(* CODESYS project motors_afag_coe.library
   Author: Miroslav Kozarev
   Placeholder: Motors_AFAG_CoE
   Title: Motors_AFAG_CoE
   Version: 0.1
   Description: Miroslav-Sashev@sensata.com
   Company: Sensata Technologies Bulgaria

Project tree, tasks and I/O mapping:
  libraries: Motors_DUTs, * (Sensata Technologies Bulgaria); Tc2_Standard, * (Beckhoff Automation GmbH); Tc3_LinMot, 1.1.0.0 (NTI AG)
  DUTs/
    Motors/
      AFAG/
        data type T_LM_Axis
        data type T_LM_DrvToPlc
  POUs/
    Motors/
      AFAG/
        Subs/
          LinMot/
            function block FB_LM_AxisControl [ST]
            function block FB_LM_MoveAbs [ST]
            function block FB_LM_MoveVelocity [ST]
            function block FB_LM_Stop [ST]
            function FN_LM_UptMCI_2 [ST]
        function block FB_ServoAxis_LinMot [ST]: A_GenOutput, A_Home, A_MoveAbsolute, A_MoveVelocity, A_ParseInput, A_ResetDone, A_SetMovementData
*)

// DUTs/Motors/AFAG/T_LM_Axis
TYPE T_LM_Axis : 
STRUCT
	PlcToDrv			AT %Q* :tstLM_PlcToDrv; 													(*PLC to Drive struct*)
	DrvToPlc			AT %I* :T_LM_DrvToPlc; 														(*Drive to PLC struct*)
	(*Status information*)
	AxisState			: tenLM_AxisState;
	CommandRunning		: BOOL;
	CommandAborted		: BOOL;
	ConfigChannelBusy	: BOOL;
	(*Information (Not required for prober work of the library function blocks)*)
	AxisName			: STRING;
	AxisNr				: UINT;
	AxisCtrlType		: STRING; 																	(*Eg. 'E1200-EC-UC', 'E1130-DP', 'B1100-GP', ....*)
END_STRUCT
END_TYPE

// DUTs/Motors/AFAG/T_LM_DrvToPlc
TYPE T_LM_DrvToPlc :
STRUCT
	StateVar 			: UINT; 																	(*StateVar of the drive*)
	StatusWord 			: UINT; 																	(*Statusword of the drive*)
	WarnWord 			: UINT; 																	(*Warnword of the drive*)
	ComDemandPosition 	: DINT; 																	(*32Bit demand position*)
	ComDemandVelocity	: DINT; 																	
	ComActualPosition 	: DINT; 																	(*32Bit actual position*)
	ComActualVelocity	: DINT; 																	

	CfgStatusWord 		: UINT;  																	(*Config Channel Status*)
	CfgIndexIn 			: UINT;  																	(*Argument (meaning depends on Cmd ID*)
	CfgValueIn 			: UDINT; 																	(*Argument (meaning depends on Cmd ID*)
END_STRUCT
END_TYPE

// POUs/Motors/AFAG/Subs/LinMot/FB_LM_AxisControl
FUNCTION_BLOCK FB_LM_AxisControl
VAR_INPUT
	SwitchOn		    : BOOL;	(*Switch on motor*)
	Home				: BOOL;	(*Start homing procedure*)
	ErrorAcknowledge	: BOOL;	(*Error acknowledge*)
	JogPlus				: BOOL;	(*Jog move postive*)
	JogMinus			: BOOL;	(*Jog move negative*)
	Band				: REAL := 10000;
END_VAR
VAR_IN_OUT
	Axis	       		: T_LM_Axis; (*Axis reference*)
END_VAR
VAR_OUTPUT
	OperationEnabled	: BOOL;	(*Axis powered on*)
	SwitchOnLocked		: BOOL;	(*Switch on locked*)
	Homed     	      	: BOOL;	(*Axis has reference*)
	MotionActive		: BOOL;	(*Motion active (Setpoint generation (VAI, curve) active)*)
	Jogging				: BOOL;	(*Axis is moving in jog mode*)
	Warning         	: BOOL;	(*Warning detected*)
	Error          		: BOOL;	(*Error detected*)
	ErrorCode      		: UINT;	(*Error code, see MotionCtrlSW manual*)
	DemandPosition  	: REAL;	(*Demand position in [mm]*)
	ActualPosition  	: REAL;	(*Actual position in [mm]*)
	ActualCurrent   	: REAL;	(*Actual motor current in [A]*)
	ActualVelocity		: REAL;
	DemandVelocity		: REAL;
END_VAR
VAR
	uiState        		: UINT;	(*internal -> Current state of the drive*)
	rTrigHome 			: LM_R_TRIG;	(*internal ->*)
	fTrigHome 			: LM_F_TRIG;	(*internal ->*)
END_VAR
(*Version history:
Date         	 | Version    		| Created under     	| Author          	| Remark 
------------------------------------------------------------------------------------------------------------------------------- 
2011-jul-12   	 | 1.0.0      		| V2.11.0 (Build 1016)	| fj  				| initial release 
2011-nov-22   	 | 1.0.1      		| V2.11.0 (Build 1016)	| fj  				| homed output reset if home input is set 
2011-dec-01   	 | 1.0.2      		| V2.11.0 (Build 1016)	| fj  				| code optimisation
2012-jan-25   	 | 1.0.3     		| V2.11.0 (Build 1016)	| fj  				| operation enabled output is now directly mapped to the status word bit 0
2012-oct-16   	 | 1.1.0      		| V2.11.0 (Build 1016)	| fj  				| added additional StateVar check for 090Fh ("homing finished") when rehoming
2014-may-13   	 | 1.0.0.1     		| v3.14014.0			| fj  				| added output DemandPosition
																				| optimized home input / homed output behaviour
*)

(*Eingänge zuweisen/lesen ][ Read and allocate inputs*)
	ActualPosition := DINT_TO_REAL(Axis.DrvToPlc.ComActualPosition)/Band;
	DemandPosition := DINT_TO_REAL(Axis.DrvToPlc.ComDemandPosition)/Band;
	ActualVelocity := DINT_TO_REAL(Axis.DrvToPlc.ComActualVelocity)/Band;
	DemandVelocity := DINT_TO_REAL(Axis.DrvToPlc.ComDemandVelocity)/Band;
	
	(*Workaround for different XML current definitions (16Bit/32Bit)*)
	//IF Axis.DrvToPlc.ComActualCurrent32 = 0 AND Axis.DrvToPlc.ComActualCurrent16 = 0 THEN
	//	ActualCurrent := 0;
	//ELSIF Axis.DrvToPlc.ComActualCurrent32 <> 0 AND Axis.DrvToPlc.ComActualCurrent16 = 0 THEN
	//	ActualCurrent := DINT_TO_REAL(Axis.DrvToPlc.ComActualCurrent32)/1000;
	//ELSIF Axis.DrvToPlc.ComActualCurrent32 = 0 AND Axis.DrvToPlc.ComActualCurrent16 <> 0 THEN
	//	ActualCurrent := INT_TO_REAL(Axis.DrvToPlc.ComActualCurrent16)/1000;
	//ELSE
	//	ActualCurrent := DINT_TO_REAL(Axis.DrvToPlc.ComActualCurrent32)/1000; (*If both 16/32Bit currents aren't 0 32Bit has higher priority*)
	//END_IF

(*Variablen ][ variables*)
	uiState := SHR(Axis.DrvToPlc.StateVar, 8);
	SwitchOnLocked := Axis.DrvToPlc.StatusWord.6;
	Warning := Axis.DrvToPlc.StatusWord.7;
	MotionActive := Axis.DrvToPlc.StatusWord.13;
	OperationEnabled := Axis.DrvToPlc.StatusWord.0;

(*=============================================================================
*  State Machine
===============================================================================*)    

CASE uiState OF
	(*Not Ready to Switch On*)
	00:	Axis.AxisState := Disabled_LM;

	(*State 4: Error*)
	04:	ErrorCode := UINT_TO_USINT(Axis.DrvToPlc.StateVar);
		Error := TRUE;
		Axis.AxisState := ErrorStop_LM;

	(*State 8: Operation Enabled*)
	08:	Homed := Axis.DrvToPlc.StateVar.7;
		IF Axis.DrvToPlc.StatusWord.13 AND NOT (Axis.AxisState = Stopping_LM) THEN
			Axis.AxisState := DiscreteMotion_LM;
		ELSIF NOT Axis.DrvToPlc.StatusWord.13 AND NOT (Axis.AxisState = Stopping_LM) THEN
			Axis.AxisState := StandStill_LM;
		END_IF

	(*State 9: Homing*)
	09:	Axis.AxisState := Homing_LM;
		IF Axis.DrvToPlc.StateVar = 16#090F THEN
			Axis.PlcToDrv.ControlWord.11 := FALSE;
		END_IF

	(*State 14: Error Behaviour QuickStop*)
	14:	Axis.AxisState := ErrorStop_LM;

	(*State 16: Jogging +*)
	16:	Axis.AxisState := Jogging_LM;

	(*State 17: Jogging -*)
	17:	Axis.AxisState := Jogging_LM;

END_CASE;


(*Wenn der drive nicht im Fehlerzustand ist, werden Error und ErrorCode auf Null gesetzt*)
(*If the drive is not in Error state, Error and ErrorCode are set to zero*)
IF uiState <> 16#04 THEN
	Error := FALSE;
	ErrorCode := 16#00;
END_IF;

IF uiState <> 16#08 THEN
	Axis.PlcToDrv.MCHeader := 16#0000; (*Reset Header to prevent "MC Cmd in wrong state" error*)
	Axis.CommandRunning := FALSE;
	Axis.CommandAborted := FALSE;
END_IF;

(*Switch On*)
Axis.PlcToDrv.ControlWord.0 := SwitchOn;
IF NOT Axis.PlcToDrv.ControlWord.0 AND NOT (uiState = 4 OR uiState = 14) THEN
	Axis.AxisState := Disabled_LM;
END_IF

(*Home*)
rTrigHome(CLK:=Home);
fTrigHome(CLK:=Home);
IF rTrigHome.Q THEN
	Axis.PlcToDrv.ControlWord.11 := TRUE;
END_IF
IF fTrigHome.Q  THEN
	Axis.PlcToDrv.ControlWord.11 := FALSE;
END_IF

IF uiState = 16#09 OR (Axis.PlcToDrv.ControlWord.11 AND NOT (uistate = 16#09)) THEN
	Homed := FALSE;
ELSE
	Homed := Axis.DrvToPlc.StatusWord.11;
END_IF

(*Error acknowledge*)
Axis.PlcToDrv.ControlWord.7 := ErrorAcknowledge;

(*JogPlus*)
Axis.PlcToDrv.ControlWord.8 := JogPlus;

(*JogMinus*)
Axis.PlcToDrv.ControlWord.9 := JogMinus;

IF (uiState = 16 OR uiState = 17) AND UINT_TO_USINT(Axis.DrvToPlc.StateVar) = 16#01 THEN
	Jogging := TRUE;
ELSE
	Jogging := FALSE;
END_IF

END_FUNCTION_BLOCK

// POUs/Motors/AFAG/Subs/LinMot/FB_LM_MoveAbs
FUNCTION_BLOCK FB_LM_MoveAbs
VAR_INPUT
	Execute			:BOOL;	(*Execute command*)
	Position		:REAL;	(*Target position in [mm]*)
	Velocity		:REAL;	(*Maximal velocity in [m/s]*)
	Acceleration	:REAL;	(*Acceleration in [m/s^2]*)
	Deceleration	:REAL;	(*Deceleration in [m/s^2]*)
	Band			: REAL := 10000;
END_VAR
VAR_IN_OUT
	Axis			:T_LM_Axis; (*Axis reference*)
	bResetDone		:BOOL;
END_VAR
VAR_OUTPUT
	Done			:BOOL;	(*Command has been executed*)
	Busy			:BOOL;	(*Command running / FB Busy*)
	Error			:BOOL;	(*Error detected*)
	ErrorID			:UINT;	(*Error ID:
							01h: Axis not ready
 							02h: Axis already has command running
 							03h: Axis has error
 							04h: Command interrupted
 							05h: Command aborted
							06h: Invalid input(s)
							*)
END_VAR

VAR_IN_OUT
	
END_VAR

VAR
	usiOldCmdCount 	:USINT;	(*internal -> *)
	usiNewCmdCount	:USINT;	(*internal -> *)
	uiCState		:UINT;	(*internal -> *)
	uiFbState		:UINT;	(*internal -> *)
	rTrig			:LM_R_TRIG;	(*internal -> *)
	udiTmpDWord		:UDINT;	(*internal -> *)

 	uiCmdHeader 	:UINT := 16#0100;	(*CommandHeader (010xh) of the "VAI Go To Position (010xh)" motion command*)
END_VAR
(*Version history:
Date         	 | Version    		| Created under     	| Author          	| Remark 
------------------------------------------------------------------------------------------------------------------------------- 
2011-jul-12   	 | 1.0.0      		| V2.11.0 (Build 1016)	| fj  				| initial release 
2011-sep-13   	 | 1.0.1      		| V2.11.0 (Build 1016)	| fj  				| removed check on "StandStill_LM"
2011-dec-01   	 | 1.0.2      		| V2.11.0 (Build 1016)	| fj  				| code optimisation
2012-apr-25   	 | 1.1.0     		| V2.11.0 (Build 1016)	| fj  				| added input parameters check
*)

(*Variablen ][ variables*)
usiOldCmdCount := SHR(UINT_TO_USINT(SHL(Axis.DrvToPlc.StateVar,4)),4);
uiCState := SHR(Axis.DrvToPlc.StateVar, 8);

IF bResetDone THEN
	Done := FALSE;
	bResetDone := FALSE;
END_IF

(*Flankenerkennung am Execute Eingang*)
(*Edge detection on Execute input*)
rTrig(CLK:=Execute);
IF rTrig.Q AND uiCState = 16#08 AND NOT Axis.CommandRunning THEN (*Start command*)
	Axis.CommandRunning := TRUE;
	Busy := TRUE;
	Done := FALSE;
	uiFbState := 1;
ELSIF rTrig.Q AND Busy THEN (*Restart command / New rising edge on execute input*)
	Axis.CommandRunning := TRUE;
	Done := FALSE;
	Busy := TRUE;
	uiFbState := 1;
ELSIF rTrig.Q AND uiCState <> 16#08 THEN (*Axis not ready*)
	uiFbState := 50; (*Error state*)
	Done := FALSE;
	Error := TRUE;
	ErrorID := 16#01; (*Axis not ready*)
ELSIF rTrig.Q AND Axis.CommandRunning AND NOT Busy THEN (*Axis already has a command running*)
	uiFbState := 50; (*Error state*)
	Error := TRUE;
	ErrorID := 16#02; (*Axis already has a command running*)
END_IF

IF Busy AND uiCState = 16#04 THEN
	Axis.CommandRunning := FALSE;
	uiFbState := 50;
	Error := TRUE;
	ErrorID := 16#03; (*Axis has error*)
END_IF

IF Busy AND uiCState <> 16#08 THEN
	Axis.CommandRunning := FALSE;
	uiFbState := 50; (*Error state*)
	Error := TRUE;
	ErrorID := 16#04; (*Command interupted*)
ELSIF Busy AND Axis.CommandAborted THEN
	uiFbState := 50; (*Error state*)
	Error := TRUE;
	ErrorID := 16#05; (*Command aborted*)
END_IF

(*State machine*)
CASE uiFbState OF
	0:	;

	1:	(*Check inputs on valid value*)
		IF (-214748.0 <= Position AND Position <= 214748.0)
			AND (0.0 < Velocity AND Velocity <= 2147.0)
			AND (0.0 < Acceleration AND Acceleration <= 21474.0)
			AND (0.0 < Deceleration AND Deceleration <= 21474.0)
			THEN
			(*Befehlskopf mit CMD Count berechen und senden ][ Calculate and send command header*)
			usiNewCmdCount := (usiOldCmdCount + 1) MOD 16 ; (*MOD 16*)
			Axis.PlcToDrv.MCHeader := 16#0000; (*Reset Header*)
			Axis.PlcToDrv.MCHeader := uiCmdHeader + usiNewCmdCount;

			udiTmpDWord := DINT_TO_UDINT(REAL_TO_DINT(Position * Band)); (*Target position*)
			Axis.PlcToDrv.MCParaWord0 := UDINT_TO_UINT(udiTmpDWord);
			Axis.PlcToDrv.MCParaWord1 := UDINT_TO_UINT(ROR(udiTmpDWord,16));

			udiTmpDWord := DINT_TO_UDINT(REAL_TO_DINT(Velocity * 100 * Band)); (*Maximal velocity*)
			Axis.PlcToDrv.MCParaWord2 := UDINT_TO_UINT(udiTmpDWord);
			Axis.PlcToDrv.MCParaWord3 := UDINT_TO_UINT(ROR(udiTmpDWord,16));

			udiTmpDWord := DINT_TO_UDINT(REAL_TO_DINT(Acceleration * 10 * Band)); (*Acceleration*)
			Axis.PlcToDrv.MCParaWord4 := UDINT_TO_UINT(udiTmpDWord);
			Axis.PlcToDrv.MCParaWord5 := UDINT_TO_UINT(ROR(udiTmpDWord,16));

			udiTmpDWord := DINT_TO_UDINT(REAL_TO_DINT(Deceleration * 10 * Band)); (*Deceleration*)
			Axis.PlcToDrv.MCParaWord6 := UDINT_TO_UINT(udiTmpDWord);
			Axis.PlcToDrv.MCParaWord7 := UDINT_TO_UINT(ROR(udiTmpDWord,16));

			FN_LM_UptMCI_2(Axis);
			
			uiFbState := 2;
		ELSE
			Axis.CommandRunning := FALSE;
			uiFbState := 50; (*Error state*)
			Error := TRUE;
			ErrorID := 16#06; (*Invalid input(s)*)
		END_IF

	2:	(*Prüfen ob Befehl ausgeführt ][ Check if command has been executed*)
		IF usiOldCmdCount = usiNewCmdCount AND uiCState = 16#08 AND Axis.DrvToPlc.StateVar.6 THEN
			Done := TRUE;
			Busy := FALSE;
			Axis.PlcToDrv.MCHeader := 16#0000 + usiNewCmdCount; (*Send no operation*)
			Axis.CommandRunning := FALSE;
			uiFbState := 3;
		END_IF

	3:	IF NOT Execute THEN
			uiFbState := 0;
			Busy := FALSE;
		END_IF

	50:	Error := TRUE;
		Busy := FALSE;
		Done := FALSE;
		IF NOT Execute THEN
			uiFbState := 0;
			Error := FALSE;
			ErrorID := 0;
		END_IF

END_CASE

END_FUNCTION_BLOCK

// POUs/Motors/AFAG/Subs/LinMot/FN_LM_UptMCI_2
FUNCTION FN_LM_UptMCI_2 : BOOL
VAR_IN_OUT
	Axis 	:T_LM_Axis;
END_VAR
VAR
END_VAR

Axis.PlcToDrv.MCParaDWord_00_03 := SHL(UINT_TO_UDINT(Axis.PlcToDrv.MCParaWord1),16) + UINT_TO_UDINT(Axis.PlcToDrv.MCParaWord0);
Axis.PlcToDrv.MCParaDWord_04_07 := SHL(UINT_TO_UDINT(Axis.PlcToDrv.MCParaWord3),16) + UINT_TO_UDINT(Axis.PlcToDrv.MCParaWord2);
Axis.PlcToDrv.MCParaDWord_08_11 := SHL(UINT_TO_UDINT(Axis.PlcToDrv.MCParaWord5),16) + UINT_TO_UDINT(Axis.PlcToDrv.MCParaWord4);
Axis.PlcToDrv.MCParaDWord_12_15 := SHL(UINT_TO_UDINT(Axis.PlcToDrv.MCParaWord7),16) + UINT_TO_UDINT(Axis.PlcToDrv.MCParaWord6);
Axis.PlcToDrv.MCParaDWord_16_19 := SHL(UINT_TO_UDINT(Axis.PlcToDrv.MCParaWord9),16) + UINT_TO_UDINT(Axis.PlcToDrv.MCParaWord8);
Axis.PlcToDrv.MCParaDWord_20_23 := SHL(UINT_TO_UDINT(Axis.PlcToDrv.MCParaWord11),16) + UINT_TO_UDINT(Axis.PlcToDrv.MCParaWord10);
Axis.PlcToDrv.MCParaDWord_24_27 := SHL(UINT_TO_UDINT(Axis.PlcToDrv.MCParaWord13),16) + UINT_TO_UDINT(Axis.PlcToDrv.MCParaWord12);

END_FUNCTION

// POUs/Motors/AFAG/Subs/LinMot/FB_LM_MoveVelocity
FUNCTION_BLOCK FB_LM_MoveVelocity
VAR_INPUT
	Execute					: BOOL;																	(*Execute command*)
	Velocity				: REAL;																	(*Maximal velocity in [m/s]*)
	Acceleration			: REAL;																	(*Acceleration in [m/s^2]*)
	NegativeDirection		: BOOL := FALSE;
	Band					: REAL := 10000;
	TargetReached			: BOOL;
END_VAR
VAR_IN_OUT
	Axis					: T_LM_Axis; 															(*Axis reference*)
END_VAR
VAR_OUTPUT
	Done					: BOOL;																	(*Command has been executed*)
	Busy					: BOOL;																	(*Command running / FB Busy*)
	Error					: BOOL;																	(*Error detected*)
	ErrorID					: UINT;																	(*Error ID:
																									01h: Axis not ready
 																									02h: Axis already has command running
 																									03h: Axis has error
 																									04h: Command interrupted
 																									05h: Command aborted
																									06h: Invalid input(s)
																									*)
END_VAR
VAR
	usiOldCmdCount 			: USINT;																(*internal -> *)
	usiNewCmdCount			: USINT;																(*internal -> *)
	uiCState				: UINT;																	(*internal -> *)
	uiFbState				: UINT;																	(*internal -> *)
	rTrig					: LM_R_TRIG;															(*internal -> *)
	udiTmpDWord				: UDINT;																(*internal -> *)

 	uiCmdHeader 			: UINT := 16#0CE0;														(*CommandHeader (0CExh) of the "VAI Dec=AccVAI Infinite Motion Positive Direction (0CExh)" motion command*)
END_VAR
(*Version history:
Date         	 | Version    		| Created under     	| Author          	| Remark 
------------------------------------------------------------------------------------------------------------------------------- 
2011-jul-12   	 | 1.0.0      		| V2.11.0 (Build 1016)	| fj  				| initial release 
2011-sep-13   	 | 1.0.1      		| V2.11.0 (Build 1016)	| fj  				| removed check for "StandStill_LM" on Execute rising edge
2011-dec-01   	 | 1.0.2      		| V2.11.0 (Build 1016)	| fj  				| code optimisation
2012-apr-25   	 | 1.1.0     		| V2.11.0 (Build 1016)	| fj  				| added input parameters check
*)

(*Variablen ][ variables*)
usiOldCmdCount := SHR(UINT_TO_USINT(SHL(Axis.DrvToPlc.StateVar,4)),4);
uiCState := SHR(Axis.DrvToPlc.StateVar, 8);

(*Flankenerkennung am Execute Eingang*)
(*Edge detection on Execute input*)
rTrig(CLK:=Execute);
IF rTrig.Q AND uiCState = 16#08 AND NOT Axis.CommandRunning THEN (*Start command*)
	Axis.CommandRunning := TRUE;
	Busy := TRUE;
	uiFbState := 1;
ELSIF rTrig.Q AND Busy THEN (*Restart command / New rising edge on execute input*)
	Axis.CommandRunning := TRUE;
	Busy := TRUE;
	uiFbState := 1;
ELSIF rTrig.Q AND uiCState <> 16#08 THEN (*Axis not ready*)
	uiFbState := 50; (*Error state*)
	Error := TRUE;
	ErrorID := 16#01; (*Axis not ready*)
ELSIF rTrig.Q AND Axis.CommandRunning AND NOT Busy THEN (*Axis already has a command running*)
	uiFbState := 50; (*Error state*)
	Error := TRUE;
	ErrorID := 16#02; (*Axis already has a command running*)
END_IF

IF Busy AND uiCState = 16#04 THEN
	Axis.CommandRunning := FALSE;
	uiFbState := 50;
	Error := TRUE;
	ErrorID := 16#03; (*Axis has error*)
END_IF

IF Busy AND uiCState <> 16#08 THEN
	Axis.CommandRunning := FALSE;
	uiFbState := 50; (*Error state*)
	Error := TRUE;
	ErrorID := 16#04; (*Command interupted*)
ELSIF Busy AND Axis.CommandAborted THEN
	uiFbState := 50; (*Error state*)
	Error := TRUE;
	ErrorID := 16#05; (*Command aborted*)
END_IF

(*State machine*)
CASE uiFbState OF
	0:	;

	1:	(*Check inputs on valid value*)
		IF (-10.0 <= ABS(Velocity) AND ABS(Velocity) <= 99999999)
			AND (0.0 < Acceleration AND Acceleration <= 99999999)
			THEN
			(*Befehlskopf mit CMD Count berechen und senden ][ Calculate and send command header*)
			usiNewCmdCount := (usiOldCmdCount + 1) MOD 16 ; (*MOD 16*)
			Axis.PlcToDrv.MCHeader := 16#0000; (*Reset Header*)
			NegativeDirection := Velocity < 0;
			IF NegativeDirection THEN
 				uiCmdHeader := 16#0CF0;
			ELSE
 				uiCmdHeader := 16#0CE0;
			END_IF
			
			Axis.PlcToDrv.MCHeader := uiCmdHeader + usiNewCmdCount;

			udiTmpDWord := DINT_TO_UDINT(REAL_TO_DINT(ABS(Velocity) * 100 * Band)); (*Maximal velocity*)
			Axis.PlcToDrv.MCParaWord0 := UDINT_TO_UINT(udiTmpDWord);
			Axis.PlcToDrv.MCParaWord1 := UDINT_TO_UINT(ROR(udiTmpDWord,16));

			udiTmpDWord := DINT_TO_UDINT(REAL_TO_DINT(Acceleration * 10000)); (*Acceleration / Deceleration*)
			Axis.PlcToDrv.MCParaWord2 := UDINT_TO_UINT(udiTmpDWord);
			Axis.PlcToDrv.MCParaWord3 := UDINT_TO_UINT(ROR(udiTmpDWord,16));
			FN_LM_UptMCI_2(Axis);

			uiFbState := 2;
		ELSE
			Axis.CommandRunning := FALSE;
			uiFbState := 50; (*Error state*)
			Error := TRUE;
			ErrorID := 16#06; (*Invalid input(s)*)
		END_IF

	2:	(*Prüfen ob Befehl ausgeführt ][ Check if command has been executed*)
		IF (usiOldCmdCount = usiNewCmdCount AND uiCState = 16#08 AND TargetReached) (*Axis.DrvToPlc.StateVar.6) OR
			TargetReached*) THEN
			Done := TRUE;
			Busy := FALSE;
			Axis.PlcToDrv.MCHeader := 16#0000 + usiNewCmdCount; (*Send no operation*)
			Axis.CommandRunning := FALSE;
			uiFbState := 3;
		END_IF

	3:	IF NOT Execute THEN
			uiFbState := 0;
			Busy := FALSE;
			Done := FALSE;
		END_IF

	50:	Error := TRUE;
		Busy := FALSE;
		Done := FALSE;
		IF NOT Execute THEN
			uiFbState := 0;
			Error := FALSE;
			ErrorID := 0;
		END_IF

END_CASE

END_FUNCTION_BLOCK

// POUs/Motors/AFAG/Subs/LinMot/FB_LM_Stop
FUNCTION_BLOCK FB_LM_Stop
VAR_INPUT
	Execute					: BOOL;																	(*Execute command*)
	Velocity				: REAL;																	(*Maximal velocity in [m/s]*)
	Acceleration			: REAL;																	(*Acceleration in [m/s^2]*)
	NegativeDirection		: BOOL := FALSE;
	Band					: REAL := 10000;
	TargetReached			: BOOL;
END_VAR
VAR_IN_OUT
	Axis					: T_LM_Axis; 															(*Axis reference*)
END_VAR
VAR_OUTPUT
	Done					: BOOL;																	(*Command has been executed*)
	Busy					: BOOL;																	(*Command running / FB Busy*)
	Error					: BOOL;																	(*Error detected*)
	ErrorID					: UINT;																	(*Error ID:
																									01h: Axis not ready
 																									02h: Axis already has command running
 																									03h: Axis has error
 																									04h: Command interrupted
 																									05h: Command aborted
																									06h: Invalid input(s)
																									*)
END_VAR
VAR
	usiOldCmdCount 			: USINT;																(*internal -> *)
	usiNewCmdCount			: USINT;																(*internal -> *)
	uiCState				: UINT;																	(*internal -> *)
	uiFbState				: UINT;																	(*internal -> *)
	rTrig					: LM_R_TRIG;															(*internal -> *)
	udiTmpDWord				: UDINT;																(*internal -> *)

 	uiCmdHeader 			: UINT := 16#0170;														(*CommandHeader (0CExh) of the "VAI Dec=AccVAI Infinite Motion Positive Direction (0CExh)" motion command*)
END_VAR
(*Version history:
Date         	 | Version    		| Created under     	| Author          	| Remark 
------------------------------------------------------------------------------------------------------------------------------- 
2011-jul-12   	 | 1.0.0      		| V2.11.0 (Build 1016)	| fj  				| initial release 
2011-sep-13   	 | 1.0.1      		| V2.11.0 (Build 1016)	| fj  				| removed check for "StandStill_LM" on Execute rising edge
2011-dec-01   	 | 1.0.2      		| V2.11.0 (Build 1016)	| fj  				| code optimisation
2012-apr-25   	 | 1.1.0     		| V2.11.0 (Build 1016)	| fj  				| added input parameters check
*)

(*Variablen ][ variables*)
usiOldCmdCount := SHR(UINT_TO_USINT(SHL(Axis.DrvToPlc.StateVar,4)),4);
uiCState := SHR(Axis.DrvToPlc.StateVar, 8);

(*Flankenerkennung am Execute Eingang*)
(*Edge detection on Execute input*)
rTrig(CLK:=Execute);
IF rTrig.Q AND uiCState = 16#08 AND NOT Axis.CommandRunning THEN (*Start command*)
	Axis.CommandRunning := TRUE;
	Busy := TRUE;
	uiFbState := 1;
ELSIF rTrig.Q AND Busy THEN (*Restart command / New rising edge on execute input*)
	Axis.CommandRunning := TRUE;
	Busy := TRUE;
	uiFbState := 1;
ELSIF rTrig.Q AND uiCState <> 16#08 THEN (*Axis not ready*)
	uiFbState := 50; (*Error state*)
	Error := TRUE;
	ErrorID := 16#01; (*Axis not ready*)
ELSIF rTrig.Q AND Axis.CommandRunning AND NOT Busy THEN (*Axis already has a command running*)
	uiFbState := 50; (*Error state*)
	Error := TRUE;
	ErrorID := 16#02; (*Axis already has a command running*)
END_IF

IF Busy AND uiCState = 16#04 THEN
	Axis.CommandRunning := FALSE;
	uiFbState := 50;
	Error := TRUE;
	ErrorID := 16#03; (*Axis has error*)
END_IF

IF Busy AND uiCState <> 16#08 THEN
	Axis.CommandRunning := FALSE;
	uiFbState := 50; (*Error state*)
	Error := TRUE;
	ErrorID := 16#04; (*Command interupted*)
ELSIF Busy AND Axis.CommandAborted THEN
	uiFbState := 50; (*Error state*)
	Error := TRUE;
	ErrorID := 16#05; (*Command aborted*)
END_IF

(*State machine*)
CASE uiFbState OF
	0:	;

	1:	(*Check inputs on valid value*)
		IF (0.0 < Acceleration AND Acceleration <= 99999999)
			THEN
			(*Befehlskopf mit CMD Count berechen und senden ][ Calculate and send command header*)
			usiNewCmdCount := (usiOldCmdCount + 1) MOD 16 ; (*MOD 16*)
			Axis.PlcToDrv.MCHeader := 16#0000; (*Reset Header*)
			
			uiCmdHeader := 16#0170;
			
			Axis.PlcToDrv.MCHeader := uiCmdHeader + usiNewCmdCount;

			udiTmpDWord := DINT_TO_UDINT(REAL_TO_DINT(Acceleration * 10000)); (*Acceleration / Deceleration*)
			Axis.PlcToDrv.MCParaWord0 := UDINT_TO_UINT(udiTmpDWord);
			Axis.PlcToDrv.MCParaWord1 := UDINT_TO_UINT(ROR(udiTmpDWord,16));
			FN_LM_UptMCI_2(Axis);

			uiFbState := 2;
		ELSE
			Axis.CommandRunning := FALSE;
			uiFbState := 50; (*Error state*)
			Error := TRUE;
			ErrorID := 16#06; (*Invalid input(s)*)
		END_IF

	2:	(*Prüfen ob Befehl ausgeführt ][ Check if command has been executed*)
		IF (usiOldCmdCount = usiNewCmdCount AND uiCState = 16#08 AND TargetReached) (*Axis.DrvToPlc.StateVar.6) OR
			TargetReached*) THEN
			Done := TRUE;
			Busy := FALSE;
			Axis.PlcToDrv.MCHeader := 16#0000 + usiNewCmdCount; (*Send no operation*)
			Axis.CommandRunning := FALSE;
			uiFbState := 3;
		END_IF

	3:	IF NOT Execute THEN
			uiFbState := 0;
			Busy := FALSE;
			Done := FALSE;
		END_IF

	50:	Error := TRUE;
		Busy := FALSE;
		Done := FALSE;
		IF NOT Execute THEN
			uiFbState := 0;
			Error := FALSE;
			ErrorID := 0;
		END_IF

END_CASE

END_FUNCTION_BLOCK

// POUs/Motors/AFAG/FB_ServoAxis_LinMot
FUNCTION_BLOCK FB_ServoAxis_LinMot																	// HJ LinMot Afaq - use with older controllers in combination with Tc3_LinMot library.
VAR_INPUT
	IsAbsolute						: BOOL := FALSE;												// Use to mark that the axis is with an absolute encoder and no homing should be executed.
	InvertMotorPolarity				: BOOL := FALSE;												// Use this to invert the motor encoder polarity from here. (CurrentPosition or TargetPosition * -1 FTW)
	Band							: REAL := 10000;												// Encoder multiplier.
	DoStop							: BOOL;															// NOT WORKING!!!
END_VAR
VAR_OUTPUT
	CurrentPosition					: LREAL;														// The current motor position.
	CurrentCommand					: UDINT;														// The current motor command.
	CurrentVelocity			 		: LREAL;														// The current motor velocity.
	Enabled							: BOOL;															// Is the motor enabled for operation.
	Error							: BOOL;															// Is the motor in an error state.
	ErrorID							: UDINT;														// If the motor is in an error state this will hold the error data.
	Moving							: BOOL;															// Is the motor moving.	
	Refferenced 					: BOOL;															// Is the motor referenced - homed.
	TraveledPath					: LREAL;														// The motor last traveled path. Currently valid only when in positioning mode.
	Busy							: BOOL;															// Is the motor busy - executing command.
	Stopped							: BOOL;															// Is the motor stopped - not working.
END_VAR
VAR_IN_OUT
	// As a test
	TargetPosition					: REAL;															// The target position of the motor. If DoMove is set in the right conditions, this will be sent to the motor.
	TargetVelocity					: REAL;															// The motor target movement velocity.
	TargetAcceleration				: REAL;															// The motor target acceleration.
	TargetDeceleration				: REAL;															// The motor target deceleration.
	TargetPrecision					: REAL;															// The motor target precision. Could use this dynamically troughout different states when the precision needs change.
	OperationMode					: UDINT := 0;													// The motor target operation mode 0 - Positioning, 1 - Velocity.
	DoServoOn						: BOOL;															// Activate the motor power up.
	DoReset							: BOOL;															// Activate the motor reset.
	DoHome							: BOOL;															// Activate the motor homing function. If the motor is marked as an absolute one this will only be reset and no homing will take place.
	DoMove							: BOOL;															// Activate a movement command. The values set in the TargetPosition, TargetVelocity and TargetAcceleration will be sent to the motor.
	TargetReached					: BOOL;															// Is the motor target reached in both modes (The target position or velocity is reached).
	axis							: T_LM_Axis;													// Lin Mot Axis reference - the actual IO structure. - LINMOT Legacy type T_LM_Axis.
END_VAR
VAR		
	state							: E_MotorStates;												// Current motor function block state.
	fbTimer							: TON;															// Used for timeouts and etc..
	fbResetTimer					: TON;															// Used for reset timeout.
	fbMoveAbsolute					: FB_LM_MoveAbs;												// Move absolute function block										- LINMOT Legacy type FB_LM_MoveAbs.
	fbMoveVelocity					: FB_LM_MoveVelocity;											// Move to velocity function block.
	fbAxisControl					: FB_LM_AxisControl;											// Axis control function block 										- LINMOT Legacy type FB_LM_AxisControl.
	fbAxisStop						: FB_LM_Stop;													// Axis stop function block.
	fbTriggerF						: F_TRIG;														// Disable trigger.
	
	PositioningMovement				: BOOL;
	VelocityMovement				: BOOL;
	
	bResetDone						: BOOL 							:= FALSE;						// Use to reset the done flag within the fbMoveAbsolute block.
	TargetTravelPath				: LREAL;														// Used to hold the target travel path.
	VelocityReached					: BOOL;
	VelocityMonitorDelimiter		: LREAL := 1000;
	TargetedVelocity				: LREAL;
	MovingToPositiong				: BOOL;
	MovingWithVelocity				: BOOL;
	MotionActive					: BOOL;
	EngageAxisStop					: BOOL;
	AxisStopping					: BOOL;
	AxisStopped						: BOOL;
	
	StopState						: DINT := 0;
	
	NegativeDirection				: BOOL := FALSE;
END_VAR

/////////////////////////////////////////////////
// NB!!!
// SET Acceleration/Deceleration at least once due to value checker. 
// 
// - prepared within the start movement state with A_SetMovementData();
//
/////////////////////////////////////////////////

//===============================================================

IF InvertMotorPolarity THEN
	TargetPosition := TargetPosition * -1;
END_IF

A_ParseInput();

fbTriggerF(CLK := DoServoOn);
		
IF fbTriggerF.Q AND 
	(state <> E_MotorStates.MOTORSTATE_ERROR) THEN
	state := E_MotorStates.MOTORSTATE_INIT;		
END_IF

IF (state <> E_MotorStates.MOTORSTATE_ERROR) AND 
	(state <> E_MotorStates.MOTORSTATE_RESET) AND 
	(state <> E_MotorStates.MOTORSTATE_ENABLE) AND 
	(DoReset = TRUE) THEN
	state := E_MotorStates.MOTORSTATE_RESET;
	IF DoMove OR 
		fbMoveAbsolute.Execute OR
		PositioningMovement OR 
		fbMoveVelocity.Execute OR
		VelocityMovement THEN
		DoMove := FALSE;
		PositioningMovement := FALSE;
		fbMoveAbsolute.Execute := FALSE;
		VelocityMovement := FALSE;
		fbMoveVelocity.Execute := FALSE;
	END_IF
	DoReset := FALSE;
END_IF

CASE state OF
	E_MotorStates.MOTORSTATE_INIT:
		DoMove := FALSE;
		PositioningMovement := FALSE;
		VelocityMovement := FALSE;
		DoHome := FALSE;
		A_ResetDone();
		DoServoOn := FALSE;
		DoReset := FALSE;
		state := E_MotorStates.MOTORSTATE_ENABLE;
		
	E_MotorStates.MOTORSTATE_ENABLE:
		IF Enabled THEN
			state := E_MotorStates.MOTORSTATE_OPERATIONAL;
		ELSIF Error OR DoReset THEN
			state := E_MotorStates.MOTORSTATE_RESET;
		END_IF
		
	E_MotorStates.MOTORSTATE_OPERATIONAL:
		IF fbTriggerF.Q THEN
			state := E_MotorStates.MOTORSTATE_INIT;	
		ELSE
			IF Error THEN
				DoServoOn := FALSE;
				state := E_MotorStates.MOTORSTATE_ERROR;
			ELSE
				IF DoMove THEN
					CASE OperationMode OF
						
						0:
							TargetReached := FALSE;
							TargetTravelPath := TargetPosition - CurrentPosition;
							A_ResetDone();
							A_SetMovementData();
							TargetedVelocity := TargetVelocity;
							//PositioningMovement := TRUE;
							StopState := 0;
							state := E_MotorStates.MOTORSTATE_MOVING;	
							
						1:
							TargetReached := FALSE;
							A_ResetDone();
							//VelocityMovement := TRUE;
							TargetedVelocity := TargetVelocity;
							NegativeDirection := TargetedVelocity < 0;
							StopState := 0;
							state := E_MotorStates.MOTORSTATE_MOVING_VELOCITY;
							
						ELSE
							
							state := E_MotorStates.MOTORSTATE_ERROR;
							
					END_CASE
				ELSIF DoHome THEN
					IF IsAbsolute THEN
						DoHome := FALSE;
					ELSE
						A_ResetDone();
						state := E_MotorStates.MOTORSTATE_HOMING;
					END_IF
				END_IF
			END_IF
		END_IF
		
	E_MotorStates.MOTORSTATE_MOVING:
		A_MoveAbsolute();
		
	E_MotorStates.MOTORSTATE_MOVING_VELOCITY:
		A_MoveVelocity();
		
	E_MotorStates.MOTORSTATE_HOMING:
		A_Home();
		
	E_MotorStates.MOTORSTATE_STOP:
		IF DoStop THEN
			EngageAxisStop := TRUE;
			fbAxisStop.Acceleration := TargetAcceleration;
			IF AxisStopped THEN
				Stopped := TRUE;
			END_IF
		ELSE
			EngageAxisStop := FALSE;
			Stopped := FALSE;
			state := E_MotorStates.MOTORSTATE_ENABLE;
		END_IF
		
	E_MotorStates.MOTORSTATE_ERROR:
		IF DoReset THEN
			IF Error THEN
				state := E_MotorStates.MOTORSTATE_RESET;
			ELSE
				state := E_MotorStates.MOTORSTATE_INIT;
			END_IF	
		END_IF
		
	E_MotorStates.MOTORSTATE_RESET:
		fbResetTimer(IN := TRUE, 
			PT := T#300MS);
		IF (NOT Error) THEN
			fbResetTimer(IN := FALSE);
			state := E_MotorStates.MOTORSTATE_INIT;
		ELSIF fbResetTimer.Q THEN
			fbResetTimer(IN := FALSE);
			DoReset := FALSE;
			state := E_MotorStates.MOTORSTATE_ERROR;
		END_IF

END_CASE

fbAxisControl(SwitchOn 					:= DoServoOn,
				Home 					:= DoHome, 
				ErrorAcknowledge 		:= DoReset,
				OperationEnabled 		=> Enabled,
				Homed 					=> Refferenced,
				MotionActive 			=> MotionActive,
				Error 					=> Error,
				ErrorCode 				=> ErrorID,
				ActualPosition 			=> CurrentPosition,
				//ActualVelocity 			=> CurrentVelocity,
				Axis 					:= axis);
				
fbMoveAbsolute(Axis 					:= axis,
				Execute 				:= PositioningMovement,
				Band					:= Band,
				Busy 					=> MovingToPositiong,
				Done 					=> TargetReached,
				bResetDone 				:= bResetDone);
				
fbAxisStop(Axis							:= axis,
	
				Execute					:= EngageAxisStop,
				
				Busy					=> AxisStopping,
				Done					=> AxisStopped);
				
				
IF OperationMode = 1 THEN
	A_GenOutput();
END_IF

fbMoveVelocity(Axis						:= axis,
				Execute					:= VelocityMovement,
				Band					:= Band,
				TargetReached			:= OperationMode = 1 AND TargetReached,
				Busy					=> MovingWithVelocity,
				Done					=> VelocityReached);
				
A_GenOutput();

IF OperationMode = 0 THEN
	Moving := MovingToPositiong OR MotionActive;
ELSE
	Moving := (ABS(CurrentVelocity) > 10) OR MovingWithVelocity;
END_IF

IF InvertMotorPolarity THEN
	CurrentPosition := CurrentPosition * -1;
END_IF

ACTION A_GenOutput:

IF VelocityMonitorDelimiter > 0 THEN
	CurrentVelocity := axis.DrvToPlc.ComActualVelocity / VelocityMonitorDelimiter;
END_IF

IF TargetPrecision > 0.0001 THEN
	IF OperationMode = 0 THEN
		TargetReached := TargetReached AND 
			(ABS(CurrentPosition - TargetPosition) < TargetPrecision) AND
			(NOT DoMove) AND
			(NOT PositioningMovement) AND
			(NOT DoStop);
	ELSIF OperationMode = 1 THEN
		IF ABS(TargetedVelocity) > 10 THEN
			TargetReached := ABS(TargetedVelocity - CurrentVelocity) < (ABS(TargetedVelocity) * (TargetPrecision / 100));
		ELSE
			TargetReached := ABS(TargetedVelocity - CurrentVelocity) < 10;
		END_IF
	END_IF
ELSE
	TargetReached := TargetReached AND 
		(ABS(CurrentPosition - TargetPosition) < 0.03) AND
		(NOT DoMove) AND
		(NOT PositioningMovement);
END_IF
END_ACTION

ACTION A_Home:
// Engage homing sequence.
IF Refferenced THEN
	DoHome := FALSE;
	state := E_MotorStates.MOTORSTATE_ENABLE;
ELSE
	IF Error THEN
		DoHome := FALSE;
		state := E_MotorStates.MOTORSTATE_ERROR;		
	END_IF
END_IF
END_ACTION

ACTION A_MoveAbsolute:
// Engage movement sequence.
IF NOT DoStop THEN
	A_SetMovementData();
END_IF
PositioningMovement := TRUE;
fbMoveAbsolute.Execute := PositioningMovement;
Busy := TRUE;
IF fbMoveAbsolute.Done AND
	(NOT DoStop) THEN
	Busy := FALSE;
	DoMove := FALSE;
	PositioningMovement := FALSE;
	fbMoveAbsolute.Execute := DoMove; 
	TraveledPath := TargetTravelPath;
	state := E_MotorStates.MOTORSTATE_ENABLE;
ELSIF fbMoveAbsolute.Error THEN
	DoMove := FALSE;
	PositioningMovement := FALSE;
	fbMoveAbsolute.Execute := DoMove;
	IF fbMoveAbsolute.ErrorID = 16#06 THEN			// BAD INPUT
		state := E_MotorStates.MOTORSTATE_RESET;
	ELSE
		Error := fbMoveAbsolute.Error;
		ErrorID := fbMoveAbsolute.ErrorID;
		state := E_MotorStates.MOTORSTATE_ERROR;
	END_IF 
ELSIF DoStop THEN
	CASE StopState OF
		0:
			fbMoveAbsolute.Execute := FALSE;
			fbMoveAbsolute.Position := CurrentPosition;
			fbMoveAbsolute.Velocity := TargetedVelocity;
			fbMoveAbsolute.Acceleration := TargetAcceleration;
			fbMoveAbsolute.Deceleration := TargetDeceleration;
			StopState := 1;
			
		1:
			fbMoveAbsolute.Position := CurrentPosition;
			fbMoveAbsolute.Velocity := TargetedVelocity;
			fbMoveAbsolute.Acceleration := TargetAcceleration;
			fbMoveAbsolute.Deceleration := TargetDeceleration;
			fbMoveAbsolute.Execute := TRUE;
			Busy := FALSE;
			DoMove := FALSE;
			PositioningMovement := FALSE;
			fbMoveAbsolute.Execute := DoMove; 
			TraveledPath := TargetTravelPath;
			state := E_MotorStates.MOTORSTATE_ENABLE;
			StopState := 2;
			
	END_CASE
END_IF
END_ACTION

ACTION A_MoveVelocity:
// Engage movement sequence.
VelocityMovement := TRUE;
fbMoveVelocity.Velocity := TargetedVelocity;
fbMoveVelocity.Acceleration := TargetAcceleration;
Busy := TRUE;
IF fbMoveVelocity.Done OR
	ABS(TargetedVelocity - CurrentVelocity) < TargetPrecision THEN
	Busy := FALSE;
	DoMove := FALSE;
	VelocityMovement := FALSE;
	TargetReached := TRUE;
	fbMoveVelocity.Execute := DoMove; 
	state := E_MotorStates.MOTORSTATE_ENABLE;
ELSIF fbMoveVelocity.Error THEN
	DoMove := FALSE;
	VelocityMovement := FALSE;
	TargetReached := FALSE;
	fbMoveVelocity.Execute := DoMove;
	IF fbMoveVelocity.ErrorID = 16#06 THEN			// BAD INPUT
		state := E_MotorStates.MOTORSTATE_RESET;
	ELSE
		Error := fbMoveVelocity.Error;
		ErrorID := fbMoveVelocity.ErrorID;
		state := E_MotorStates.MOTORSTATE_ERROR;
	END_IF 
END_IF
END_ACTION

ACTION A_ParseInput:
// Parse axis input data.

fbAxisControl(  
	Band				:= Band,
	OperationEnabled 	=> Enabled,
	Homed 				=> Refferenced,
	MotionActive 		=> Moving,
	Error 				=> Error,
	ErrorCode 			=> ErrorID,
	ActualPosition 		=> CurrentPosition,
	//ActualVelocity 		=> CurrentVelocity,
	Axis 				:= axis);
END_ACTION

ACTION A_ResetDone:
// USE THIS TO RESET THE Done (TargetReached act.)

bResetDone := TRUE;
END_ACTION

ACTION A_SetMovementData:
// Set the movement data for the movement block.

fbMoveAbsolute.Position := TargetPosition;
fbMoveAbsolute.Velocity := TargetedVelocity;
fbMoveAbsolute.Acceleration := TargetAcceleration;
fbMoveAbsolute.Deceleration := TargetDeceleration;
END_ACTION

END_FUNCTION_BLOCK
